(* CODESYS project Traslo_st_UBICA_POR_COLOR_y_ROBOT+TABLA-.project
   CompiledLibraryCompatibilityVersion: CODESYS V3.5 SP16 Patch 4

Project tree, tasks and I/O mapping:
  Device : CODESYS Control Win V3 x64, 3S - Smart Software Solutions GmbH, version 3.5.16.40
    application Application
      libraries: Standard, * (System); VisuDialogs, * (System); CmpBitmapPool, * (System)
      task VISU_TASK (cyclic, interval 100 ms, priority 31) calls VisuElems.Visu_Prg
      task MainTask (cyclic, interval t#20ms, priority 1) calls PLC_PRG
      program ANALOGICAS [LD]
      Symbols
      program PLC_PRG [ST]
      visualisation Panel_control
      global variables GVL
      function block ESCALADO [FBD]
      image pool ImagePool
  libraries: Util, * (System); Net Base Services, 3.5.19.20 (3S - Smart Software Solutions GmbH)
  5ce3da45-db07-42e7-a21c-a00fff4ed8f6|C:\Users\GGARCES\OneDrive - congeladosnavarra.com\ICONOS\scada\SETA_EMERG_ON.png
  text list GlobalTextList
  5ce3da45-db07-42e7-a21c-a00fff4ed8f6|C:\Users\GGARCES\OneDrive - congeladosnavarra.com\ICONOS\scada\SETA_EMERG_OFF.png
*)

// Device/Application/GVL
{attribute 'qualified_only'}
VAR_GLOBAL
	VISION_AZUL : BOOL;
	VISION_VERDE : BOOL;
	VISION_METAL : BOOL;
	NUMERO_ESTANTE : REAL;
	POSICION : REAL;
	x_position : REAL;                          //max 9 posiciones
	Z_position : REAL;
	X_position_FILTRADA: REAL;
	Z_position_FILTRADA: REAL;
END_VAR

// Device/Application/PLC_PRG
PROGRAM PLC_PRG
VAR
	Tim_carga : TON ; 
	sys_on: BOOL;
	sys_auto: BOOL;
	sys_man: BOOL;
	count : INT;
	count_forks: INT;
	flanco_carga: BOOL;flanco_forks_out: BOOL;
	R_TRIG1: R_trig;R_TRIG : R_TRIG;
	R_TRIG_ESTANTE : R_TRIG;
	CTU_MOV: CTU;
	TIM_POSICION: TOF;
	Tim_descarga: TON;
	TRASLO_CARGADO: BOOL;
	TIM_POS0: TON;
	Tim_descarga1: TON;
	PALET_POS: BOOL;
	Tim_descarga2: TON;
	Tim_descarga3: TON;
	Tim_descarga4: TON;
	Tim_descarga5: TON;
	R_TRIG_AZUL: R_TRIG;
	R_TRIG_VERDE: R_TRIG;
	R_TRIG_METAL: R_TRIG;
	CTU_AZUL: CTU;
	CTU_VERDE : CTU;
	CTU_METAL : CTU;
	CNT_TOTAL : CTU;
	CNT_PIEZAS : CTU;
	// color verde
	pos1 : BOOL;
	pos2 : BOOL;
	pos3 : BOOL;
	pos4 : BOOL;
	pos5 : BOOL;
	pos6 : BOOL;
	pos7 : BOOL;
	pos8 : BOOL;
	pos9 : BOOL;
	pos10 : BOOL;
	pos11 : BOOL;
	pos12 : BOOL;	
    pos13 : BOOL;
	pos14 : BOOL;
	pos15 : BOOL;
	pos16 : BOOL;
	pos17 : BOOL;
	pos18 : BOOL;
	// color azul
	pos19 : BOOL;
	pos20 : BOOL;
	pos21 : BOOL;
	pos22 : BOOL;
	pos23 : BOOL;
	pos24 : BOOL;
	pos25 : BOOL;
	pos26 : BOOL;
	pos27 : BOOL;
	pos28 : BOOL;
	pos29 : BOOL;
	pos30 : BOOL;	
    pos31 : BOOL;
	pos32 : BOOL;
	pos33 : BOOL;
	pos34 : BOOL;
	pos35 : BOOL;
	pos36 : BOOL;
	// color metal
	pos37 : BOOL;
	pos38 : BOOL;
	pos39 : BOOL;
	pos40 : BOOL;
	pos41 : BOOL;
	pos42 : BOOL;
	pos43 : BOOL;
	pos44 : BOOL;
	pos45 : BOOL;
	pos46 : BOOL;
	pos47 : BOOL;
	pos48 : BOOL;	
    pos49 : BOOL;
	pos50 : BOOL;
	pos51 : BOOL;
	pos52 : BOOL;
	pos53 : BOOL;
	pos54 : BOOL;
	
	color_verde_saturado : BOOL;
	color_azul_saturado : BOOL;
	color_metal_saturado : BOOL;
	SENSOR0_0: BOOL;
	TON_bajar1 : ton ;
	TON_subir1 : ton ;
	TON_bajar2 : ton ;
	TON_subir2 : ton ;
	TON_avanzar : ton ;
	TON_retroceder : ton ;
	TON_reset: ton;
	fin_ciclo_robot_cartesiano : BOOL ;
	a: BOOL;
	bit1 : INT ;
	CONTADOR_TOTAL: WORD;
	REGISTRO: ARRAY [1..55] OF WORD;
	POS: word;
	STARTFP: r_trig;
END_VAR
VAR_INPUT
	At_entry : BOOL;
	At_exit : BOOL;
	At_load : BOOL;
	At_unload : BOOL;
	SENSOR_0: BOOL;
	SENSOR_1: BOOL;
	auto : BOOL;
	Emergency_stop : BOOL;
	Manual : BOOL;
	limit_right : BOOL;
	limit_left : BOOL;
	Reset : BOOL;
	Start : BOOL;
	Stop : BOOL;
	stacker_crane_limit_right : BOOL;
	stacker_crane_limit_left : BOOL;
	stacker_crane_limit_middle : BOOL;
	MANDAR_POSICION : BOOL;
	GO: BOOL;
	RESET_NUMERO_ESTANTE : BOOL;
	SENSOR_piezas_cinta :BOOL;
	robot_ocupado : BOOL;
	FALLO_ROBOT : BOOL;
	detec_piezas_cartesiano : BOOL ;
	deteccion_pieza_robot_cart: BOOL;
END_VAR

VAR_OUTPUT
	//rodillos
	Emitter : BOOL;
	RODILLOS_1: BOOL;
	CURVA_RODILLOS_2: BOOL;
	RODILLOS_3: BOOL;
	Entry_CONVEYOR_3 : BOOL;
	Load_conveyor_4 : BOOL;
	Exit_conveyor : BOOL;
	UnLoad_conveyor_4 : BOOL;
	Remover : BOOL;
	
	Forks_left : BOOL;
	Forks_right : BOOL;
	// luces
	Reset_light : BOOL;
	Start_light : BOOL;
	Stop_light : BOOL;
	
	stacker_crane_x_sp : REAL;
	stacker_crane_z_sp : REAL;
	ALARMA_ACTIVA : BOOL;
	
	Emisor_piezas : BOOL;
	cinta_piezas : BOOL;
	ON_ROBOT : BOOL ;
	
	bajar_robot_cartesiano : BOOL;
	subir_robot_cartesiano : BOOL;
	agarrar_pieza_robot_cart : BOOL ;
	avanzar_robot_cartesiano : BOOL ;
	
	CINTA_PIEZAS_ACABADAS : BOOL ;
	TOPE_PIEZAS : BOOL ;
END_VAR


ANALOGICAS ();

// PROGRAMA PARA SIMULAR CON FACTORY IO UN TRASLO

//emergencia
IF NOT Emergency_stop OR NOT Stop THEN
	sys_on := FALSE;
	sys_auto:= FALSE;
	Entry_CONVEYOR_3 := FALSE;
	Load_conveyor_4 := FALSE;
	Forks_left := FALSE;
	Forks_right := FALSE;
	stacker_crane_x_sp := 0;
    stacker_crane_z_sp := 0;
	TRASLO_CARGADO := FALSE;
	COUNT_FORKS := 0;
	gvl.Z_position := 0;
	gvl.x_position := 0;
	PALET_POS := FALSE;
	GVL.POSICION := 0;
	pos1 := 0;pos2 := 0;pos3 := 0;pos4 := 0;pos5 := 0;pos6 := 0;pos7 := 0;pos8 := 0;pos9 := 0;pos10:= 0;
	pos11:= 0;pos12:= 0;pos13:= 0;pos14:= 0;pos15:= 0;pos16:= 0;pos17:= 0;pos18:= 0;pos19:= 0;pos20:= 0;
	pos21:= 0;pos22:= 0;pos23:= 0;pos24:= 0;pos25:= 0;pos26:= 0;pos27:= 0;pos28:= 0;pos29:= 0;pos30:= 0;
	pos31:= 0;pos32:= 0;pos33:= 0;pos34:= 0;pos35:= 0;pos36:= 0;pos37:= 0;pos38:= 0;pos39:= 0;pos40:= 0;
	pos41:= 0;pos42:= 0;pos43:= 0;pos44:= 0;pos45:= 0;pos46:= 0;pos47:= 0;pos48:= 0;pos49:= 0;pos50:= 0;
	pos51:= 0;pos52:= 0;pos53:= 0;pos54:= 0;
	POS:=0;
    
END_IF

// FALLO POSICION 0 EN FACTORY I/O FILTRO PARA QUE FUNCIONE BIEN
IF gvl.X_position_FILTRADA <0 THEN gvl.X_position_FILTRADA :=0;
IF gvl.Z_position_FILTRADA <0 THEN gvl.Z_position_FILTRADA :=0;	
END_IF
END_IF

// On
IF Start AND auto THEN
	sys_on := TRUE;
	stacker_crane_x_sp := 0;
    stacker_crane_z_sp := 0;
END_IF

//Auto
IF sys_on AND auto THEN
	sys_auto:= TRUE;
	sys_man := FALSE;
END_IF

// Manual
IF sys_on AND manual THEN
	sys_auto:= FALSE;
	sys_man := TRUE;
END_IF

// Reset
IF reset  THEN
	count:= 0;
	count_forks := 0;
	stacker_crane_x_sp := 0;
    stacker_crane_z_sp := 0;
	GVL.POSICION := 0;
END_IF

IF RESET AND NOT stacker_crane_limit_middle AND stacker_crane_limit_left THEN Forks_right := TRUE; END_IF
IF RESET AND NOT stacker_crane_limit_middle AND stacker_crane_limit_right THEN Forks_left := TRUE; END_IF 
IF RESET AND stacker_crane_limit_middle THEN 
	Forks_right := FALSE;
	Forks_left := FALSE;
    PALET_POS := FALSE;	
END_IF

// EMISOR DE PALETS
IF SYS_ON AND SENSOR_0 AND NOT ALARMA_ACTIVA THEN
	Emitter := TRUE;
END_IF
IF Emitter AND NOT SENSOR_0 OR NOT SYS_ON THEN
	Emitter := false;
END_IF
// Caminos de rodillos 1
IF sys_auto AND bit1 = 8 AND CURVA_RODILLOS_2  AND NOT ALARMA_ACTIVA AND NOT Emitter THEN
	RODILLOS_1 := TRUE;
END_IF	
IF sys_auto AND NOT CURVA_RODILLOS_2 OR Emitter OR  ALARMA_ACTIVA THEN
	RODILLOS_1 := FALSE;
END_IF
// Curva de rodillos 2
IF sys_auto AND RODILLOS_3 AND NOT ALARMA_ACTIVA THEN
	CURVA_RODILLOS_2 := TRUE;
IF sys_auto AND NOT SENSOR_1 AND NOT ALARMA_ACTIVA OR NOT RODILLOS_3 THEN
	CURVA_RODILLOS_2 := FALSE;
END_IF
END_IF
// Caminos de rodillos 3
IF sys_auto AND Entry_CONVEYOR_3 AND NOT ALARMA_ACTIVA THEN
	RODILLOS_3 := TRUE;
END_IF
IF sys_auto AND NOT at_entry AND NOT ALARMA_ACTIVA OR NOT Entry_CONVEYOR_3 THEN
    RODILLOS_3 := FALSE;
END_IF
// Entry conveyor 3
IF sys_auto AND Load_conveyor_4 AND NOT ALARMA_ACTIVA THEN
	Entry_CONVEYOR_3 := TRUE;
END_IF
IF sys_auto AND NOT at_load AND NOT ALARMA_ACTIVA OR NOT Load_conveyor_4 THEN
    Entry_CONVEYOR_3 := FALSE;
END_IF
// load conveyor 4
IF sys_auto AND at_load AND NOT ALARMA_ACTIVA THEN
	Load_conveyor_4 := TRUE;
ELSE
	Load_conveyor_4 := FALSE;	
END_IF

// Flanco contador palets a traslo
    R_TRIG(CLK:= NOT At_load, Q=> flanco_carga); 

// Llamada a traslo y asigna posicion 
IF FLANCO_CARGA THEN
	Entry_CONVEYOR_3 := FALSE;
	Load_conveyor_4 := FALSE;
END_IF
// TIEMPO EN POSICION DE INICIO
	TIM_POS0(IN := gvl.x_position_FILTRADA < 0.1 AND gvl.Z_position_FILTRADA =0 AND NOT AT_LOAD , PT:= T#1S); 
	IF TIM_POS0.Q THEN
	PALET_POS := TRUE;
	else
	PALET_POS:= FALSE;
	END_IF

// CONTROL DE PALETS POR PRODUCTO -----COLOR------

R_TRIG_AZUL(CLK:= GVL.VISION_AZUL);
R_TRIG_VERDE(CLK:= GVL.VISION_VERDE);
R_TRIG_METAL(CLK:= GVL.VISION_METAL);

CTU_AZUL(CU:= R_TRIG_AZUL.CLK, RESET:=RESET OR NOT Emergency_stop);
CTU_VERDE(CU:= R_TRIG_VERDE.CLK, RESET:=RESET OR NOT Emergency_stop);
CTU_METAL(CU:= R_TRIG_METAL.CLK, RESET:=RESET OR NOT Emergency_stop);

//AZUL
IF R_TRIG_AZUL.CLK THEN 
	GVL.POSICION := CTU_AZUL.CV;
END_IF
//VERDE
IF R_TRIG_VERDE.CLK THEN 
	GVL.POSICION := CTU_VERDE.CV + 18;
END_IF
//METAL
IF R_TRIG_METAL.CLK THEN 
	GVL.POSICION := CTU_METAL.CV + 36;
END_IF
// ------------ COGER PALET ---------------
// salida uñas
IF PALET_POS AND stacker_crane_limit_middle THEN
	Forks_left := TRUE;
END_IF

IF flanco_forks_out THEN
	count_forks := count_forks + 1;
END_IF

//FLANCO_UÑAS CARGA FUERA
R_TRIG1(CLK:=Forks_left AND NOT stacker_crane_limit_middle, Q=> flanco_forks_out); 

// RETARDO RECOGIDA UÑAS
Tim_carga(IN := stacker_crane_limit_left, PT:= T#1S); 

// elevar coger palet
IF stacker_crane_limit_left AND sys_auto AND stacker_crane_x_sp = 0 (*atras*)THEN
	stacker_crane_z_sp :=0.30;
END_IF

// uñas atras
IF stacker_crane_limit_left AND stacker_crane_z_sp >= 0.3 AND Tim_carga.Q THEN
	Forks_left := FALSE;
	TRASLO_CARGADO := TRUE;
	PALET_POS := FALSE;
END_IF 

// contador de palets en el traslo     
CTU_MOV(CU:= stacker_crane_limit_middle AND count_forks = 1 AND NOT MANDAR_POSICION AND NOT GO, RESET:=RESET OR RESET_NUMERO_ESTANTE OR NOT Emergency_stop, PV:= 100); 
CNT_TOTAL(CU:= count_forks = 1,RESET:= RESET AND NOT Emergency_stop,PV:= 55);
//
TIM_POSICION(IN := count_forks = 1 AND stacker_crane_limit_middle, PT:= T#200S); 
// RESET CONTADOR CUANDO ELIGES ESTANTERIA EN MANUAL
R_TRIG_ESTANTE (CLK:= RESET_NUMERO_ESTANTE );

//-----------------------------------------------------------------------------


//------------ PRIMERA FILA --------------------------


//-----------------------------------------------------------------------------
// POSICION 1
IF GVL.POSICION = 1 AND count_forks=1 AND stacker_crane_limit_middle AND TIM_POSICION.Q THEN
     stacker_crane_x_sp := 1.06;
     stacker_crane_z_sp := 0.8;
END_IF
// dejar carga posicion 1
IF GVL.POSICION = 1 AND TIM_POSICION.Q AND count_forks=1 AND gvl.x_position_FILTRADA < 0.98 AND gvl.x_position_FILTRADA > 0.96 AND gvl.Z_position_FILTRADA < 0.8 AND gvl.Z_position_FILTRADA > 0.7 THEN 
    Forks_right := TRUE;	
IF stacker_crane_limit_right THEN
	stacker_crane_z_sp := 0.4;
END_IF	
END_IF
//-----------------------------------------------------------------------------

// POSICION 2
IF GVL.POSICION = 2 AND count_forks=1 AND stacker_crane_limit_middle AND TIM_POSICION.Q THEN
	 stacker_crane_x_sp := 2.14;
     stacker_crane_z_sp := 0.8;
END_IF 
// dejar carga posicion 2
IF GVL.POSICION = 2 AND TIM_POSICION.Q AND count_forks=1 AND gvl.x_position_FILTRADA < 2.07 AND gvl.x_position_FILTRADA > 2.05 AND gvl.Z_position_FILTRADA < 0.8 AND gvl.Z_position_FILTRADA > 0.7 THEN 
    Forks_right := TRUE;
IF stacker_crane_limit_right THEN
	stacker_crane_z_sp := 0.4;
END_IF	
END_IF

//-----------------------------------------------------------------------------
// POSICION 3
IF GVL.POSICION = 3 AND count_forks=1 AND stacker_crane_limit_middle AND TIM_POSICION.Q THEN
	  stacker_crane_x_sp := 3.21;
     stacker_crane_z_sp := 0.8;
END_IF 
// dejar carga posicion 3
IF GVL.POSICION = 3 AND TIM_POSICION.Q AND count_forks=1 AND gvl.x_position < 3.22 AND gvl.x_position > 3.20 AND gvl.Z_position < 0.8 AND gvl.Z_position > 0.7 THEN 
    Forks_right := TRUE;
IF stacker_crane_limit_right THEN
	stacker_crane_z_sp := 0.4;
END_IF	
END_IF  
//-----------------------------------------------------------------------------

// POSICION 4
IF GVL.POSICION = 4 AND count_forks=1 AND stacker_crane_limit_middle AND TIM_POSICION.Q THEN
	  stacker_crane_x_sp := 4.28;
     stacker_crane_z_sp := 0.8;
	 END_IF
// dejar carga posicion 4
IF GVL.POSICION = 4 AND TIM_POSICION.Q AND count_forks=1 AND gvl.x_position < 4.29 AND gvl.x_position > 4.27 AND gvl.Z_position < 0.8 AND gvl.Z_position > 0.7 THEN 
    Forks_right := TRUE;
IF stacker_crane_limit_right THEN
	stacker_crane_z_sp := 0.4;
	
END_IF  
END_IF 
//-----------------------------------------------------------------------------
// POSICION 5
IF GVL.POSICION = 5 AND count_forks=1 AND stacker_crane_limit_middle AND TIM_POSICION.Q THEN
	  stacker_crane_x_sp := 5.36;
     stacker_crane_z_sp := 0.8;
END_IF 
// dejar carga posicion 5
IF GVL.POSICION = 5 AND TIM_POSICION.Q AND count_forks=1 AND gvl.x_position < 5.37 AND gvl.x_position > 5.35 AND gvl.Z_position < 0.8 AND gvl.Z_position > 0.7 THEN 
    Forks_right := TRUE;
IF stacker_crane_limit_right THEN
	stacker_crane_z_sp := 0.4;	
END_IF  
END_IF
//-----------------------------------------------------------------------------
// POSICION 6
IF GVL.POSICION = 6 AND count_forks=1 AND stacker_crane_limit_middle AND TIM_POSICION.Q THEN
	  stacker_crane_x_sp := 6.45;
     stacker_crane_z_sp := 0.8;
END_IF 
// dejar carga posicion 6
IF GVL.POSICION = 6 AND TIM_POSICION.Q AND count_forks=1 AND gvl.x_position < 6.46 AND gvl.x_position > 6.44 AND gvl.Z_position < 0.9 AND gvl.Z_position > 0.7 THEN 
    Forks_right := TRUE;
IF stacker_crane_limit_right THEN
	stacker_crane_z_sp := 0.4;
END_IF  
END_IF 
//-----------------------------------------------------------------------------
// POSICION 7
IF GVL.POSICION = 7 AND count_forks=1 AND stacker_crane_limit_middle AND TIM_POSICION.Q THEN
	  stacker_crane_x_sp := 7.52;
     stacker_crane_z_sp := 0.8;
END_IF 
// dejar carga posicion 7
IF GVL.POSICION = 7 AND TIM_POSICION.Q AND count_forks=1 AND gvl.x_position < 7.53 AND gvl.x_position > 7.51 AND gvl.Z_position < 0.9 AND gvl.Z_position > 0.7 THEN 
    Forks_right := TRUE;
IF stacker_crane_limit_right THEN
	stacker_crane_z_sp := 0.4;
END_IF	
END_IF  
//-----------------------------------------------------------------------------
// POSICION 8
IF GVL.POSICION = 8 AND count_forks=1 AND stacker_crane_limit_middle AND TIM_POSICION.Q THEN
	  stacker_crane_x_sp := 8.59;
     stacker_crane_z_sp := 0.8;
END_IF 
// dejar carga posicion 8
IF GVL.POSICION = 8 AND TIM_POSICION.Q AND count_forks=1 AND gvl.x_position < 8.60 AND gvl.x_position > 8.58 AND gvl.Z_position < 0.9 AND gvl.Z_position > 0.7 THEN 
    Forks_right := TRUE;
IF stacker_crane_limit_right THEN
	stacker_crane_z_sp := 0.4;
END_IF	
END_IF  
//-----------------------------------------------------------------------------
// POSICION 9
IF GVL.POSICION = 9 AND count_forks=1 AND stacker_crane_limit_middle AND TIM_POSICION.Q THEN
	  stacker_crane_x_sp := 9.66;
     stacker_crane_z_sp := 0.8;
END_IF 
// dejar carga posicion 9
IF GVL.POSICION = 9 AND TIM_POSICION.Q AND count_forks=1 AND gvl.x_position > 9.65 AND gvl.x_position < 9.67 AND gvl.Z_position < 0.9 AND gvl.Z_position > 0.7 THEN 
    Forks_right := TRUE;
IF stacker_crane_limit_right THEN
	stacker_crane_z_sp := 0.4;
END_IF	
END_IF  
//-----------------------------------------------------------------------------

// --------- SEGUNDA FILA --------------


//-----------------------------------------------------------------------------

// POSICION 10
IF GVL.POSICION = 10 AND count_forks=1 AND stacker_crane_limit_middle AND TIM_POSICION.Q  THEN
	  stacker_crane_x_sp := 1.06;
      stacker_crane_z_sp := 2.50;
END_IF 
// dejar carga posicion 10
IF GVL.POSICION = 10 AND TIM_POSICION.Q AND count_forks=1 AND gvl.x_position < 1.07 AND gvl.x_position > 1.05 AND gvl.Z_position < 2.51 AND gvl.Z_position > 2.49 THEN 
    Forks_right := TRUE;
IF stacker_crane_limit_right THEN
	stacker_crane_z_sp := 2.0;
END_IF	
END_IF  
//-----------------------------------------------------------------------------

// POSICION 11
IF GVL.POSICION = 11 AND count_forks=1 AND stacker_crane_limit_middle AND TIM_POSICION.Q  THEN
	  stacker_crane_x_sp := 2.15;
      stacker_crane_z_sp := 2.5;
END_IF 
// dejar carga posicion 11
IF GVL.POSICION = 11 AND TIM_POSICION.Q AND count_forks=1 AND gvl.x_position < 2.16 AND gvl.x_position > 2.14 AND gvl.Z_position < 2.51 AND gvl.Z_position > 2.49 THEN 
    Forks_right := TRUE;
IF stacker_crane_limit_right THEN
	stacker_crane_z_sp := 2.0;
END_IF	
END_IF  
//-----------------------------------------------------------------------------

// POSICION 12
IF GVL.POSICION = 12 AND count_forks=1 AND stacker_crane_limit_middle AND TIM_POSICION.Q  THEN
	  stacker_crane_x_sp := 3.21;
      stacker_crane_z_sp := 2.5;
END_IF 
// dejar carga posicion 12
IF GVL.POSICION = 12 AND TIM_POSICION.Q AND count_forks=1 AND gvl.x_position < 3.22 AND gvl.x_position > 3.20 AND gvl.Z_position < 2.51 AND gvl.Z_position > 2.49 THEN 
    Forks_right := TRUE;
IF stacker_crane_limit_right THEN
	stacker_crane_z_sp := 2.0;
END_IF	
END_IF  
//-----------------------------------------------------------------------------

// POSICION 13
IF GVL.POSICION = 13 AND count_forks=1 AND stacker_crane_limit_middle AND TIM_POSICION.Q  THEN
	  stacker_crane_x_sp := 4.28;
      stacker_crane_z_sp := 2.5;
END_IF 
// dejar carga posicion 13
IF GVL.POSICION = 13 AND TIM_POSICION.Q AND count_forks=1 AND gvl.x_position < 4.29 AND gvl.x_position > 4.27 AND gvl.Z_position < 2.51 AND gvl.Z_position > 2.49 THEN 
    Forks_right := TRUE;
IF stacker_crane_limit_right THEN
	stacker_crane_z_sp := 2.0;
END_IF	
END_IF  
//-----------------------------------------------------------------------------

// POSICION 14
IF GVL.POSICION = 14 AND count_forks=1 AND stacker_crane_limit_middle AND TIM_POSICION.Q  THEN
	  stacker_crane_x_sp := 5.36;
      stacker_crane_z_sp := 2.5;
END_IF 
// dejar carga posicion 14
IF GVL.POSICION = 14 AND TIM_POSICION.Q AND count_forks=1 AND gvl.x_position < 5.37 AND gvl.x_position > 5.35 AND gvl.Z_position < 2.51 AND gvl.Z_position > 2.49 THEN 
    Forks_right := TRUE;
IF stacker_crane_limit_right THEN
	stacker_crane_z_sp := 2.0;
END_IF	
END_IF  
//-----------------------------------------------------------------------------

// POSICION 15
IF GVL.POSICION = 15 AND count_forks=1 AND stacker_crane_limit_middle AND TIM_POSICION.Q  THEN
	  stacker_crane_x_sp := 6.45;
      stacker_crane_z_sp := 2.5;
END_IF 
// dejar carga posicion 15
IF GVL.POSICION = 15 AND TIM_POSICION.Q AND count_forks=1 AND gvl.x_position < 6.46 AND gvl.x_position > 6.44 AND gvl.Z_position < 2.51 AND gvl.Z_position > 2.49 THEN 
    Forks_right := TRUE;
IF stacker_crane_limit_right THEN
	stacker_crane_z_sp := 2.0;
END_IF	
END_IF  
//-----------------------------------------------------------------------------

// POSICION 16
IF GVL.POSICION = 16 AND count_forks=1 AND stacker_crane_limit_middle AND TIM_POSICION.Q  THEN
	  stacker_crane_x_sp := 7.52;
      stacker_crane_z_sp := 2.5;
END_IF 
// dejar carga posicion 16
IF GVL.POSICION = 16 AND TIM_POSICION.Q AND count_forks=1 AND gvl.x_position < 7.53 AND gvl.x_position > 7.51 AND gvl.Z_position < 2.51 AND gvl.Z_position > 2.49 THEN 
    Forks_right := TRUE;
IF stacker_crane_limit_right THEN
	stacker_crane_z_sp := 2.0;
END_IF	
END_IF  
//-----------------------------------------------------------------------------

// POSICION 17
IF GVL.POSICION = 17 AND count_forks=1 AND stacker_crane_limit_middle AND TIM_POSICION.Q  THEN
	  stacker_crane_x_sp := 8.59;
      stacker_crane_z_sp := 2.5;
END_IF 
// dejar carga posicion 17
IF GVL.POSICION = 17 AND TIM_POSICION.Q AND count_forks=1 AND gvl.x_position < 8.60 AND gvl.x_position > 8.58 AND gvl.Z_position < 2.51 AND gvl.Z_position > 2.49 THEN 
    Forks_right := TRUE;
IF stacker_crane_limit_right THEN
	stacker_crane_z_sp := 2.0;
END_IF	
END_IF  
//-----------------------------------------------------------------------------

// POSICION 18
IF GVL.POSICION = 18 AND count_forks=1 AND stacker_crane_limit_middle AND TIM_POSICION.Q  THEN
	  stacker_crane_x_sp := 9.66;
      stacker_crane_z_sp := 2.5;
END_IF 
// dejar carga posicion 18
IF GVL.POSICION = 18 AND TIM_POSICION.Q AND count_forks=1 AND gvl.x_position < 9.67 AND gvl.x_position > 9.65 AND gvl.Z_position < 2.51 AND gvl.Z_position > 2.49 THEN 
    Forks_right := TRUE;
IF stacker_crane_limit_right THEN
	stacker_crane_z_sp := 2.0;
END_IF	
END_IF  
//-----------------------------------------------------------------------------  

// --------- TERCERA FILA --------------

//-----------------------------------------------------------------------------
// POSICION 19
IF GVL.POSICION = 19 AND count_forks=1 AND stacker_crane_limit_middle AND TIM_POSICION.Q  THEN
	  stacker_crane_x_sp := 1.06;
      stacker_crane_z_sp := 4.20;
END_IF 
// dejar carga posicion 19
IF GVL.POSICION = 19 AND TIM_POSICION.Q AND count_forks=1 AND gvl.x_position < 1.07 AND gvl.x_position > 1.05 AND gvl.Z_position < 4.21 AND gvl.Z_position > 4.19 THEN 
    Forks_right := TRUE;
IF stacker_crane_limit_right THEN
	stacker_crane_z_sp := 3.90;
END_IF	
END_IF  
//-----------------------------------------------------------------------------

// POSICION 20
IF GVL.POSICION = 20 AND count_forks=1 AND stacker_crane_limit_middle AND TIM_POSICION.Q  THEN
	  stacker_crane_x_sp := 2.15;
      stacker_crane_z_sp := 4.20;
END_IF 
// dejar carga posicion 20
IF GVL.POSICION = 20 AND TIM_POSICION.Q AND count_forks=1 AND gvl.x_position < 2.16 AND gvl.x_position > 2.14 AND gvl.Z_position < 4.21 AND gvl.Z_position > 4.19 THEN 
    Forks_right := TRUE;
IF stacker_crane_limit_right THEN
	stacker_crane_z_sp := 3.90;
END_IF	
END_IF  
//-----------------------------------------------------------------------------

// POSICION 21
IF GVL.POSICION = 21 AND count_forks=1 AND stacker_crane_limit_middle AND TIM_POSICION.Q  THEN
	  stacker_crane_x_sp := 3.21;
      stacker_crane_z_sp := 4.20;
END_IF 
// dejar carga posicion 21
IF GVL.POSICION = 21 AND TIM_POSICION.Q AND count_forks=1 AND gvl.x_position < 3.22 AND gvl.x_position > 3.20 AND gvl.Z_position < 4.21 AND gvl.Z_position > 4.19 THEN 
    Forks_right := TRUE;
IF stacker_crane_limit_right THEN
	stacker_crane_z_sp := 3.90;
END_IF	
END_IF  
//-----------------------------------------------------------------------------

// POSICION 22
IF GVL.POSICION = 22 AND count_forks=1 AND stacker_crane_limit_middle AND TIM_POSICION.Q  THEN
	  stacker_crane_x_sp := 4.29;
      stacker_crane_z_sp := 4.20;
END_IF 
// dejar carga posicion 22
IF GVL.POSICION = 22 AND TIM_POSICION.Q AND count_forks=1 AND gvl.x_position < 4.30 AND gvl.x_position > 4.28 AND gvl.Z_position < 4.21 AND gvl.Z_position > 4.19 THEN 
    Forks_right := TRUE;
IF stacker_crane_limit_right THEN
	stacker_crane_z_sp := 3.90;
END_IF	
END_IF  
//-----------------------------------------------------------------------------

// POSICION 23
IF GVL.POSICION = 23 AND count_forks=1 AND stacker_crane_limit_middle AND TIM_POSICION.Q  THEN
	  stacker_crane_x_sp := 5.36;
      stacker_crane_z_sp := 4.20;
END_IF 
// dejar carga posicion 23
IF GVL.POSICION = 23 AND TIM_POSICION.Q AND count_forks=1 AND gvl.x_position < 5.37 AND gvl.x_position > 5.35 AND gvl.Z_position < 4.21 AND gvl.Z_position > 4.19 THEN 
    Forks_right := TRUE;
IF stacker_crane_limit_right THEN
	stacker_crane_z_sp := 3.90;
END_IF	
END_IF  
//-----------------------------------------------------------------------------

// POSICION 24
IF GVL.POSICION = 24 AND count_forks=1 AND stacker_crane_limit_middle AND TIM_POSICION.Q  THEN
	  stacker_crane_x_sp := 6.44;
      stacker_crane_z_sp := 4.20;
END_IF 
// dejar carga posicion 24
IF GVL.POSICION = 24 AND TIM_POSICION.Q AND count_forks=1 AND gvl.x_position < 6.45 AND gvl.x_position > 6.43 AND gvl.Z_position < 4.21 AND gvl.Z_position > 4.19 THEN 
    Forks_right := TRUE;
IF stacker_crane_limit_right THEN
	stacker_crane_z_sp := 3.90;
END_IF	
END_IF  
//-----------------------------------------------------------------------------

// POSICION 25
IF GVL.POSICION = 25 AND count_forks=1 AND stacker_crane_limit_middle AND TIM_POSICION.Q  THEN
	  stacker_crane_x_sp := 7.51;
      stacker_crane_z_sp := 4.20;
END_IF 
// dejar carga posicion 25
IF GVL.POSICION = 25 AND TIM_POSICION.Q AND count_forks=1 AND gvl.x_position < 7.52 AND gvl.x_position > 7.50 AND gvl.Z_position < 4.21 AND gvl.Z_position > 4.19 THEN 
    Forks_right := TRUE;
IF stacker_crane_limit_right THEN
	stacker_crane_z_sp := 3.90;
END_IF	
END_IF  
//-----------------------------------------------------------------------------

// POSICION 26
IF GVL.POSICION = 26 AND count_forks=1 AND stacker_crane_limit_middle AND TIM_POSICION.Q  THEN
	  stacker_crane_x_sp := 8.59;
      stacker_crane_z_sp := 4.20;
END_IF 
// dejar carga posicion 26
IF GVL.POSICION = 26 AND TIM_POSICION.Q AND count_forks=1 AND gvl.x_position < 8.60 AND gvl.x_position > 8.58 AND gvl.Z_position < 4.21 AND gvl.Z_position > 4.19 THEN 
    Forks_right := TRUE;
IF stacker_crane_limit_right THEN
	stacker_crane_z_sp := 3.90;
END_IF	
END_IF  
//-----------------------------------------------------------------------------

// POSICION 27
IF GVL.POSICION = 27 AND count_forks=1 AND stacker_crane_limit_middle AND TIM_POSICION.Q  THEN
	  stacker_crane_x_sp := 9.66;
      stacker_crane_z_sp := 4.20;
END_IF 
// dejar carga posicion 27
IF GVL.POSICION = 27 AND TIM_POSICION.Q AND count_forks=1 AND gvl.x_position < 9.67 AND gvl.x_position > 9.65 AND gvl.Z_position < 4.21 AND gvl.Z_position > 4.19 THEN 
    Forks_right := TRUE;
IF stacker_crane_limit_right THEN
	stacker_crane_z_sp := 3.90;
END_IF	
END_IF  
//-----------------------------------------------------------------------------  


// --------- CUARTA FILA --------------

//-----------------------------------------------------------------------------
// POSICION 28
IF GVL.POSICION = 28 AND count_forks=1 AND stacker_crane_limit_middle AND TIM_POSICION.Q  THEN
	  stacker_crane_x_sp := 1.06;
      stacker_crane_z_sp := 5.66;
END_IF 
// dejar carga posicion 28
IF GVL.POSICION = 28 AND TIM_POSICION.Q AND count_forks=1 AND gvl.x_position < 1.07 AND gvl.x_position > 1.05 AND gvl.Z_position < 5.67 AND gvl.Z_position > 5.65 THEN 
    Forks_right := TRUE;
IF stacker_crane_limit_right THEN
	stacker_crane_z_sp := 5.40;
END_IF	
END_IF  
//-----------------------------------------------------------------------------

// POSICION 29
IF GVL.POSICION = 29 AND count_forks=1 AND stacker_crane_limit_middle AND TIM_POSICION.Q  THEN
	  stacker_crane_x_sp := 2.15;
      stacker_crane_z_sp := 5.66;
END_IF 
// dejar carga posicion 29
IF GVL.POSICION = 29 AND TIM_POSICION.Q AND count_forks=1 AND gvl.x_position < 2.16 AND gvl.x_position > 2.14 AND gvl.Z_position < 5.67 AND gvl.Z_position > 5.65 THEN 
    Forks_right := TRUE;
IF stacker_crane_limit_right THEN
	stacker_crane_z_sp := 5.40;
END_IF	
END_IF  
//-----------------------------------------------------------------------------

// POSICION 30
IF GVL.POSICION = 30 AND count_forks=1 AND stacker_crane_limit_middle AND TIM_POSICION.Q  THEN
	  stacker_crane_x_sp := 3.21;
      stacker_crane_z_sp := 5.66;
END_IF 
// dejar carga posicion 30
IF GVL.POSICION = 30 AND TIM_POSICION.Q AND count_forks=1 AND gvl.x_position < 3.22 AND gvl.x_position > 3.20 AND gvl.Z_position < 5.67 AND gvl.Z_position > 5.65 THEN 
    Forks_right := TRUE;
IF stacker_crane_limit_right THEN
	stacker_crane_z_sp := 5.40;
END_IF	
END_IF  
//-----------------------------------------------------------------------------

// POSICION 31
IF GVL.POSICION = 31 AND count_forks=1 AND stacker_crane_limit_middle AND TIM_POSICION.Q  THEN
	  stacker_crane_x_sp := 4.29;
      stacker_crane_z_sp := 5.66;
END_IF 
// dejar carga posicion 31
IF GVL.POSICION = 31 AND TIM_POSICION.Q AND count_forks=1 AND gvl.x_position < 4.30 AND gvl.x_position > 4.28 AND gvl.Z_position < 5.67 AND gvl.Z_position > 5.65 THEN 
    Forks_right := TRUE;
IF stacker_crane_limit_right THEN
	stacker_crane_z_sp := 5.40;
END_IF	
END_IF  
//-----------------------------------------------------------------------------

// POSICION 32
IF GVL.POSICION = 32 AND count_forks=1 AND stacker_crane_limit_middle AND TIM_POSICION.Q  THEN
	  stacker_crane_x_sp := 5.36;
      stacker_crane_z_sp := 5.66;
END_IF 
// dejar carga posicion 32
IF GVL.POSICION = 32 AND TIM_POSICION.Q AND count_forks=1 AND gvl.x_position < 5.37 AND gvl.x_position > 5.35 AND gvl.Z_position < 5.67 AND gvl.Z_position > 5.65 THEN 
    Forks_right := TRUE;
IF stacker_crane_limit_right THEN
	stacker_crane_z_sp := 5.40;
END_IF	
END_IF  
//-----------------------------------------------------------------------------

// POSICION 33
IF GVL.POSICION = 33 AND count_forks=1 AND stacker_crane_limit_middle AND TIM_POSICION.Q  THEN
	  stacker_crane_x_sp := 6.45;
      stacker_crane_z_sp := 5.66;
END_IF 
// dejar carga posicion 33
IF GVL.POSICION = 33 AND TIM_POSICION.Q AND count_forks=1 AND gvl.x_position < 6.46 AND gvl.x_position > 6.44 AND gvl.Z_position < 5.67 AND gvl.Z_position > 5.65 THEN 
    Forks_right := TRUE;
IF stacker_crane_limit_right THEN
	stacker_crane_z_sp := 5.40;
END_IF	
END_IF  
//-----------------------------------------------------------------------------

// POSICION 34
IF GVL.POSICION = 34 AND count_forks=1 AND stacker_crane_limit_middle AND TIM_POSICION.Q  THEN
	  stacker_crane_x_sp := 7.51;
      stacker_crane_z_sp := 5.66;
END_IF 
// dejar carga posicion 34
IF GVL.POSICION = 34 AND TIM_POSICION.Q AND count_forks=1 AND gvl.x_position < 7.52 AND gvl.x_position > 7.50 AND gvl.Z_position < 5.67 AND gvl.Z_position > 5.65 THEN 
    Forks_right := TRUE;
IF stacker_crane_limit_right THEN
	stacker_crane_z_sp := 5.40;
END_IF	
END_IF  
//-----------------------------------------------------------------------------

// POSICION 35
IF GVL.POSICION = 35 AND count_forks=1 AND stacker_crane_limit_middle AND TIM_POSICION.Q  THEN
	  stacker_crane_x_sp := 8.59;
      stacker_crane_z_sp := 5.66;
END_IF 
// dejar carga posicion 35
IF GVL.POSICION = 35 AND TIM_POSICION.Q AND count_forks=1 AND gvl.x_position < 8.60 AND gvl.x_position > 8.58 AND gvl.Z_position < 5.67 AND gvl.Z_position > 5.65 THEN 
    Forks_right := TRUE;
IF stacker_crane_limit_right THEN
	stacker_crane_z_sp := 5.40;
END_IF	
END_IF  
//-----------------------------------------------------------------------------

// POSICION 36
IF GVL.POSICION = 36 AND count_forks=1 AND stacker_crane_limit_middle AND TIM_POSICION.Q  THEN
	  stacker_crane_x_sp := 9.66;
      stacker_crane_z_sp := 5.66;
END_IF 
// dejar carga posicion 36
IF GVL.POSICION = 36 AND TIM_POSICION.Q AND count_forks=1 AND gvl.x_position < 9.67 AND gvl.x_position > 9.65 AND gvl.Z_position < 5.67 AND gvl.Z_position > 5.65 THEN 
    Forks_right := TRUE;
IF stacker_crane_limit_right THEN
	stacker_crane_z_sp := 5.40;
END_IF	
END_IF 
//-----------------------------------------------------------------------------  

// --------- QUINTA FILA --------------

//-----------------------------------------------------------------------------
// POSICION 37
IF GVL.POSICION = 37 AND count_forks=1 AND stacker_crane_limit_middle AND TIM_POSICION.Q  THEN
	  stacker_crane_x_sp := 1.06;
      stacker_crane_z_sp := 7.50;
END_IF 
// dejar carga posicion 37
IF GVL.POSICION = 37 AND TIM_POSICION.Q AND count_forks=1 AND gvl.x_position < 1.07 AND gvl.x_position > 1.05 AND gvl.Z_position < 7.51 AND gvl.Z_position > 7.49 THEN 
    Forks_right := TRUE;
IF stacker_crane_limit_right THEN
	stacker_crane_z_sp := 7.30;
END_IF	
END_IF  
//-----------------------------------------------------------------------------

// POSICION 38
IF GVL.POSICION = 38 AND count_forks=1 AND stacker_crane_limit_middle AND TIM_POSICION.Q  THEN
	  stacker_crane_x_sp := 2.15;
      stacker_crane_z_sp := 7.50;
END_IF 
// dejar carga posicion 38
IF GVL.POSICION = 38 AND TIM_POSICION.Q AND count_forks=1 AND gvl.x_position < 2.16 AND gvl.x_position > 2.14 AND gvl.Z_position < 7.51 AND gvl.Z_position > 7.49 THEN 
    Forks_right := TRUE;
IF stacker_crane_limit_right THEN
	stacker_crane_z_sp := 7.30;
END_IF	
END_IF  
//-----------------------------------------------------------------------------

// POSICION 39
IF GVL.POSICION = 39 AND count_forks=1 AND stacker_crane_limit_middle AND TIM_POSICION.Q  THEN
	  stacker_crane_x_sp := 3.21;
      stacker_crane_z_sp := 7.50;
END_IF 
// dejar carga posicion 39
IF GVL.POSICION = 39 AND TIM_POSICION.Q AND count_forks=1 AND gvl.x_position < 3.22 AND gvl.x_position > 3.20 AND gvl.Z_position < 7.51 AND gvl.Z_position > 7.49 THEN 
    Forks_right := TRUE;
IF stacker_crane_limit_right THEN
	stacker_crane_z_sp := 7.30;
END_IF	
END_IF  
//-----------------------------------------------------------------------------

// POSICION 40
IF GVL.POSICION = 40 AND count_forks=1 AND stacker_crane_limit_middle AND TIM_POSICION.Q  THEN
	  stacker_crane_x_sp := 4.29;
      stacker_crane_z_sp := 7.50;
END_IF 
// dejar carga posicion 40
IF GVL.POSICION = 40 AND TIM_POSICION.Q AND count_forks=1 AND gvl.x_position < 4.30 AND gvl.x_position > 4.28 AND gvl.Z_position < 7.51 AND gvl.Z_position > 7.49 THEN 
    Forks_right := TRUE;
IF stacker_crane_limit_right THEN
	stacker_crane_z_sp := 7.30;
END_IF	
END_IF  
//-----------------------------------------------------------------------------

// POSICION 41
IF GVL.POSICION = 41 AND count_forks=1 AND stacker_crane_limit_middle AND TIM_POSICION.Q  THEN
	  stacker_crane_x_sp := 5.36;
      stacker_crane_z_sp := 7.50;
END_IF 
// dejar carga posicion 41
IF GVL.POSICION = 41 AND TIM_POSICION.Q AND count_forks=1 AND gvl.x_position < 5.37 AND gvl.x_position > 5.35 AND gvl.Z_position < 7.51 AND gvl.Z_position > 7.49 THEN 
    Forks_right := TRUE;
IF stacker_crane_limit_right THEN
	stacker_crane_z_sp := 7.30;
END_IF	
END_IF  
//-----------------------------------------------------------------------------

// POSICION 42
IF GVL.POSICION = 42 AND count_forks=1 AND stacker_crane_limit_middle AND TIM_POSICION.Q  THEN
	  stacker_crane_x_sp := 6.45;
      stacker_crane_z_sp := 7.50;
END_IF 
// dejar carga posicion 42
IF GVL.POSICION = 42 AND TIM_POSICION.Q AND count_forks=1 AND gvl.x_position < 6.46 AND gvl.x_position > 6.44 AND gvl.Z_position < 7.51 AND gvl.Z_position > 7.49 THEN 
    Forks_right := TRUE;
IF stacker_crane_limit_right THEN
	stacker_crane_z_sp := 7.30;
END_IF	
END_IF  
//-----------------------------------------------------------------------------

// POSICION 43
IF GVL.POSICION = 43 AND count_forks=1 AND stacker_crane_limit_middle AND TIM_POSICION.Q  THEN
	  stacker_crane_x_sp := 7.51;
      stacker_crane_z_sp := 7.50;
END_IF 
// dejar carga posicion 43
IF GVL.POSICION = 43 AND TIM_POSICION.Q AND count_forks=1 AND gvl.x_position < 7.52 AND gvl.x_position > 7.50 AND gvl.Z_position < 7.51 AND gvl.Z_position > 7.49 THEN 
    Forks_right := TRUE;
IF stacker_crane_limit_right THEN
	stacker_crane_z_sp := 7.30;
END_IF	
END_IF  
//-----------------------------------------------------------------------------

// POSICION 44
IF GVL.POSICION = 44 AND count_forks=1 AND stacker_crane_limit_middle AND TIM_POSICION.Q  THEN
	  stacker_crane_x_sp := 8.59;
      stacker_crane_z_sp := 7.50;
END_IF 
// dejar carga posicion 44
IF GVL.POSICION = 44 AND TIM_POSICION.Q AND count_forks=1 AND gvl.x_position < 8.60 AND gvl.x_position > 8.58 AND gvl.Z_position < 7.51 AND gvl.Z_position > 7.49 THEN 
    Forks_right := TRUE;
IF stacker_crane_limit_right THEN
	stacker_crane_z_sp := 7.30;
END_IF	
END_IF  
//-----------------------------------------------------------------------------

// POSICION 45
IF GVL.POSICION = 45 AND count_forks=1 AND stacker_crane_limit_middle AND TIM_POSICION.Q  THEN
	  stacker_crane_x_sp := 9.66;
      stacker_crane_z_sp := 7.50;
END_IF 
// dejar carga posicion 45
IF GVL.POSICION = 45 AND TIM_POSICION.Q AND count_forks=1 AND gvl.x_position < 9.67 AND gvl.x_position > 9.65 AND gvl.Z_position < 7.51 AND gvl.Z_position > 7.49 THEN 
    Forks_right := TRUE;
IF stacker_crane_limit_right THEN
	stacker_crane_z_sp := 7.30;
END_IF	
END_IF 
//----------------------------------------------------------------------------- 

// --------- SEXTA FILA --------------

//-----------------------------------------------------------------------------
// POSICION 46
IF GVL.POSICION = 46 AND count_forks=1 AND stacker_crane_limit_middle AND TIM_POSICION.Q  THEN
	  stacker_crane_x_sp := 1.06;
      stacker_crane_z_sp := 9.20;
END_IF 
// dejar carga posicion 46
IF GVL.POSICION = 46 AND TIM_POSICION.Q AND count_forks=1 AND gvl.x_position < 1.07 AND gvl.x_position > 1.05 AND gvl.Z_position < 9.21 AND gvl.Z_position > 9.19 THEN 
    Forks_right := TRUE;
IF stacker_crane_limit_right THEN
	stacker_crane_z_sp := 9.0;
END_IF	
END_IF  
//-----------------------------------------------------------------------------

// POSICION 47
IF GVL.POSICION = 47 AND count_forks=1 AND stacker_crane_limit_middle AND TIM_POSICION.Q  THEN
	  stacker_crane_x_sp := 2.15;
      stacker_crane_z_sp := 9.20;
END_IF 
// dejar carga posicion 47
IF GVL.POSICION = 47 AND TIM_POSICION.Q AND count_forks=1 AND gvl.x_position < 2.16 AND gvl.x_position > 2.14 AND gvl.Z_position < 9.21 AND gvl.Z_position > 9.19 THEN 
    Forks_right := TRUE;
IF stacker_crane_limit_right THEN
	stacker_crane_z_sp := 9.0;
END_IF	
END_IF  
//-----------------------------------------------------------------------------

// POSICION 48
IF GVL.POSICION = 48 AND count_forks=1 AND stacker_crane_limit_middle AND TIM_POSICION.Q  THEN
	  stacker_crane_x_sp := 3.21;
      stacker_crane_z_sp := 9.20;
END_IF 
// dejar carga posicion 48
IF GVL.POSICION = 48 AND TIM_POSICION.Q AND count_forks=1 AND gvl.x_position < 3.22 AND gvl.x_position > 3.20 AND gvl.Z_position < 9.21 AND gvl.Z_position > 9.19 THEN 
    Forks_right := TRUE;
IF stacker_crane_limit_right THEN
	stacker_crane_z_sp := 9.0;
END_IF	
END_IF  
//-----------------------------------------------------------------------------

// POSICION 49
IF GVL.POSICION = 49 AND count_forks=1 AND stacker_crane_limit_middle AND TIM_POSICION.Q  THEN
	  stacker_crane_x_sp := 4.29;
      stacker_crane_z_sp := 9.20;
END_IF 
// dejar carga posicion 49
IF GVL.POSICION = 49 AND TIM_POSICION.Q AND count_forks=1 AND gvl.x_position < 4.30 AND gvl.x_position > 4.28 AND gvl.Z_position < 9.21 AND gvl.Z_position > 9.19 THEN 
    Forks_right := TRUE;
IF stacker_crane_limit_right THEN
	stacker_crane_z_sp := 9.0;
END_IF	
END_IF  
//-----------------------------------------------------------------------------

// POSICION 50
IF GVL.POSICION = 50 AND count_forks=1 AND stacker_crane_limit_middle AND TIM_POSICION.Q  THEN
	  stacker_crane_x_sp := 5.36;
      stacker_crane_z_sp := 9.20;
END_IF 
// dejar carga posicion 50
IF GVL.POSICION = 50 AND TIM_POSICION.Q AND count_forks=1 AND gvl.x_position < 5.37 AND gvl.x_position > 5.35 AND gvl.Z_position < 9.21 AND gvl.Z_position > 9.19 THEN 
    Forks_right := TRUE;
IF stacker_crane_limit_right THEN
	stacker_crane_z_sp := 9.0;
END_IF	
END_IF  
//-----------------------------------------------------------------------------

// POSICION 51
IF GVL.POSICION = 51 AND count_forks=1 AND stacker_crane_limit_middle AND TIM_POSICION.Q  THEN
	  stacker_crane_x_sp := 6.45;
      stacker_crane_z_sp := 9.20;
END_IF 
// dejar carga posicion 51
IF GVL.POSICION = 51 AND TIM_POSICION.Q AND count_forks=1 AND gvl.x_position < 6.46 AND gvl.x_position > 6.44 AND gvl.Z_position < 9.21 AND gvl.Z_position > 9.19 THEN 
    Forks_right := TRUE;
IF stacker_crane_limit_right THEN
	stacker_crane_z_sp := 9.0;
END_IF	
END_IF  
//-----------------------------------------------------------------------------

// POSICION 52
IF GVL.POSICION = 52 AND count_forks=1 AND stacker_crane_limit_middle AND TIM_POSICION.Q  THEN
	  stacker_crane_x_sp := 7.51;
      stacker_crane_z_sp := 9.20;
END_IF 
// dejar carga posicion 52
IF GVL.POSICION = 52 AND TIM_POSICION.Q AND count_forks=1 AND gvl.x_position < 7.52 AND gvl.x_position > 7.50 AND gvl.Z_position < 9.21 AND gvl.Z_position > 9.19 THEN 
    Forks_right := TRUE;
IF stacker_crane_limit_right THEN
	stacker_crane_z_sp := 9.0;
END_IF	
END_IF  
//-----------------------------------------------------------------------------

// POSICION 53
IF GVL.POSICION = 53 AND count_forks=1 AND stacker_crane_limit_middle AND TIM_POSICION.Q  THEN
	  stacker_crane_x_sp := 8.59;
      stacker_crane_z_sp := 9.20;
END_IF 
// dejar carga posicion 53
IF GVL.POSICION = 53 AND TIM_POSICION.Q AND count_forks=1 AND gvl.x_position < 8.60 AND gvl.x_position > 8.58 AND gvl.Z_position < 9.21 AND gvl.Z_position > 9.19 THEN 
    Forks_right := TRUE;
IF stacker_crane_limit_right THEN
	stacker_crane_z_sp := 9.0;
END_IF	
END_IF  
//-----------------------------------------------------------------------------

// POSICION 54
IF GVL.POSICION = 54 AND count_forks=1 AND stacker_crane_limit_middle AND TIM_POSICION.Q  THEN
	  stacker_crane_x_sp := 9.66;
      stacker_crane_z_sp := 9.20;
END_IF 
// dejar carga posicion 54
IF GVL.POSICION = 54 AND TIM_POSICION.Q AND count_forks=1 AND gvl.x_position < 9.67 AND gvl.x_position > 9.65 AND gvl.Z_position < 9.21 AND gvl.Z_position > 9.19 THEN 
    Forks_right := TRUE;
IF stacker_crane_limit_right THEN
	stacker_crane_z_sp := 9.0;
END_IF	
END_IF 
//----------------------------------------------------------------------------- 


//---------------- RECOGER UÑA Y VOLVER A INICIO----------------------------------- 



//-----------------------------------------------------------------------------
	// RETARDO RECOGIDA UÑAS ABAJO
    Tim_descarga(IN := stacker_crane_limit_right AND stacker_crane_z_sp < 0.41 AND stacker_crane_z_sp > 0.39 , PT:= T#1S);
IF Tim_descarga.Q	THEN
	Forks_right := FALSE;
	count_forks := 0;
END_IF	
IF MANDAR_POSICION AND TIM_DESCARGA.Q THEN
	RESET_NUMERO_ESTANTE := TRUE;
END_IF

	// RETARDO RECOGIDA UÑAS SEGUNDA ALTURA
    Tim_descarga1(IN := stacker_crane_limit_right AND stacker_crane_z_sp < 2.01 AND stacker_crane_z_sp > 1.99 , PT:= T#1S);
IF Tim_descarga1.Q	THEN
	Forks_right := FALSE;
	count_forks := 0;
END_IF
IF MANDAR_POSICION AND TIM_DESCARGA1.Q THEN
	RESET_NUMERO_ESTANTE := TRUE;
END_IF

	// RETARDO RECOGIDA UÑAS TERCERA ALTURA
    Tim_descarga2(IN := stacker_crane_limit_right AND stacker_crane_z_sp < 3.91 AND stacker_crane_z_sp > 3.89, PT:= T#1S);
IF Tim_descarga2.Q	THEN
	Forks_right := FALSE;
	count_forks := 0;
END_IF
IF MANDAR_POSICION AND TIM_DESCARGA2.Q THEN
	RESET_NUMERO_ESTANTE := TRUE;
END_IF

	// RETARDO RECOGIDA UÑAS CUARTA ALTURA
    Tim_descarga3(IN := stacker_crane_limit_right AND stacker_crane_z_sp < 5.41 AND stacker_crane_z_sp > 5.39, PT:= T#1S);
IF Tim_descarga3.Q	THEN
	Forks_right := FALSE;
	count_forks := 0;
END_IF
IF MANDAR_POSICION AND TIM_DESCARGA3.Q THEN
	RESET_NUMERO_ESTANTE := TRUE;
END_IF

    // RETARDO RECOGIDA UÑAS QUINTA ALTURA
    Tim_descarga4(IN := stacker_crane_limit_right AND stacker_crane_z_sp < 7.31 AND stacker_crane_z_sp > 7.29, PT:= T#1S);
IF Tim_descarga4.Q	THEN
	Forks_right := FALSE;
	count_forks := 0;
END_IF
IF MANDAR_POSICION AND TIM_DESCARGA4.Q THEN
	RESET_NUMERO_ESTANTE := TRUE;
END_IF

    // RETARDO RECOGIDA UÑAS SEXTA ALTURA
    Tim_descarga5(IN := stacker_crane_limit_right AND stacker_crane_z_sp < 9.01 AND stacker_crane_z_sp > 8.99, PT:= T#1S);
IF Tim_descarga5.Q	THEN
	Forks_right := FALSE;
	count_forks := 0;
END_IF
IF MANDAR_POSICION AND TIM_DESCARGA5.Q THEN
	RESET_NUMERO_ESTANTE := TRUE;
END_IF

// VUELTA DESDE UBICACION DE DESCARGA EN ESTANTERIA A UBICACION DE CARGA
IF NOT FORKS_RIGHT AND COUNT_FORKS =0 AND stacker_crane_limit_middle AND TRASLO_CARGADO THEN
	TRASLO_CARGADO := FALSE;
    stacker_crane_x_sp := 0;
    stacker_crane_Z_sp := 0;
	CTU_MOV.RESET := FALSE;
END_IF

//-------- VISUALIZACION UBICACION EN INSTRUMENTACION DEL CUADRO-------------
  GVL.NUMERO_ESTANTE := CTU_MOV.CV;
  
//-------- ocupacion de estanterias color azul-----------
STARTFP(CLK:= flanco_forks_out );

IF gvl.POSICION = 1 AND startfp.Q THEN
pos1:= 1; 
pos := POS + 1;
REGISTRO[POS] := 1;
END_IF
IF gvl.POSICION = 2 AND startfp.Q THEN
pos2:= 1;
POS := POS + 1;
REGISTRO[POS] := 2;
END_IF
IF gvl.POSICION = 3 AND startfp.Q THEN 
pos3:= 1;
POS := POS + 1;
REGISTRO[POS] := 3;
END_IF
IF gvl.POSICION = 4 AND startfp.Q THEN
pos4:= 1;
pos := POS + 1;
REGISTRO[POS] := 4;
END_IF
IF gvl.POSICION = 5 AND startfp.Q THEN
pos5:= 1;
pos := POS + 1;
REGISTRO[POS] := 5;
END_IF
IF gvl.POSICION = 6 AND startfp.Q THEN
pos6:= 1;
pos := POS + 1;
REGISTRO[POS] := 6;
END_IF
IF gvl.POSICION = 7 AND startfp.Q THEN
pos7:= 1;
pos := POS + 1;
REGISTRO[POS] := 7;
END_IF
IF gvl.POSICION = 8 AND startfp.Q THEN
pos8:= 1;
pos := POS + 1;
REGISTRO[POS] := 8;
END_IF
IF gvl.POSICION = 9 AND startfp.Q THEN
pos9:= 1;
pos := POS + 1;
REGISTRO[POS] := 9;
END_IF
IF gvl.POSICION = 10 AND startfp.Q THEN
pos10:= 1;
pos := POS + 1;
REGISTRO[POS] := 10;
END_IF
IF gvl.POSICION = 11 AND startfp.Q THEN
pos11:= 1;
pos := POS + 1;
REGISTRO[POS] := 11;
END_IF
IF gvl.POSICION = 12 AND startfp.Q THEN
pos12:= 1;
pos := POS + 1;
REGISTRO[POS] := 12;
END_IF
IF gvl.POSICION = 13 AND startfp.Q THEN 
pos13:= 1;
pos := POS + 1;
REGISTRO[POS] := 13;
END_IF
IF gvl.POSICION = 14 AND startfp.Q THEN
pos14:= 1;
pos := POS + 1;
REGISTRO[POS] := 14;
END_IF
IF gvl.POSICION = 15 AND startfp.Q THEN
pos15:= 1;
pos := POS + 1;
REGISTRO[POS] := 15;
END_IF
IF gvl.POSICION = 16 AND startfp.Q THEN
pos16:= 1;
pos := POS + 1;
REGISTRO[POS] := 16;
END_IF
IF gvl.POSICION = 17 AND startfp.Q THEN
pos17:= 1;
pos := POS + 1;
REGISTRO[POS] := 17;
END_IF
IF gvl.POSICION = 18 AND startfp.Q THEN
pos18:= 1; 
pos := POS + 1;
REGISTRO[POS] := 18;
END_IF

//-------- ocupacion de estanterias color verde-----------
IF gvl.POSICION = 19 AND startfp.Q THEN
pos19:= 1;
pos := POS + 1;
REGISTRO[POS] := 19;
END_IF
IF gvl.POSICION = 20 AND startfp.Q THEN
pos20:= 1;
pos := POS + 1;
REGISTRO[POS] := 20;
END_IF
IF gvl.POSICION = 21 AND startfp.Q THEN
pos21:= 1;
pos := POS + 1;
REGISTRO[POS] := 21;
END_IF
IF gvl.POSICION = 22 AND startfp.Q THEN
pos22:= 1;
pos := POS + 1;
REGISTRO[POS] := 22;
END_IF
IF gvl.POSICION = 23 AND startfp.Q THEN
pos23:= 1;
pos := POS + 1;
REGISTRO[POS] := 23;
END_IF
IF gvl.POSICION = 24 AND startfp.Q THEN
pos24:= 1;
pos := POS + 1;
REGISTRO[POS] := 24;
END_IF
IF gvl.POSICION = 25 AND startfp.Q THEN
pos25:= 1;
pos := POS + 1;
REGISTRO[POS] := 25;
END_IF
IF gvl.POSICION = 26 AND startfp.Q THEN
pos26:= 1;
pos := POS + 1;
REGISTRO[POS] := 26;
END_IF
IF gvl.POSICION = 27 AND startfp.Q THEN
pos27:= 1;
pos := POS + 1;
REGISTRO[POS] := 27;
END_IF
IF gvl.POSICION = 28 AND startfp.Q THEN
pos28:= 1;
pos := POS + 1;
REGISTRO[POS] := 28;
END_IF
IF gvl.POSICION = 29 AND startfp.Q THEN
pos29:= 1;
pos := POS + 1;
REGISTRO[POS] := 29;
END_IF
IF gvl.POSICION = 30 AND startfp.Q THEN
pos30:= 1;
pos := POS + 1;
REGISTRO[POS] := 30;
END_IF
IF gvl.POSICION = 31 AND startfp.Q THEN
pos31:= 1;
pos := POS + 1;
REGISTRO[POS] := 31;
END_IF
IF gvl.POSICION = 32 AND startfp.Q THEN
pos32:= 1;
pos := POS + 1;
REGISTRO[POS] := 32;
END_IF
IF gvl.POSICION = 33 AND startfp.Q THEN
pos33:= 1;
pos := POS + 1;
REGISTRO[POS] := 33;
END_IF
IF gvl.POSICION = 34 AND startfp.Q THEN
pos34:= 1;
pos := POS + 1;
REGISTRO[POS] := 34;
END_IF
IF gvl.POSICION = 35 AND startfp.Q THEN
pos35:= 1;
pos := POS + 1;
REGISTRO[POS] := 35;
END_IF
IF gvl.POSICION = 36 AND startfp.Q THEN
pos36:= 1;
pos := POS + 1;
REGISTRO[POS] := 36;
END_IF

//-------- ocupacion de estanterias color metal-----------
IF gvl.POSICION = 37 AND startfp.Q THEN
pos37:= 1;
pos := POS + 1;
REGISTRO[POS] := 37;
END_IF
IF gvl.POSICION = 38 AND startfp.Q THEN
pos38:= 1;
pos := POS + 1;
REGISTRO[POS] := 38;
END_IF
IF gvl.POSICION = 39 AND startfp.Q THEN
pos39:= 1;
pos := POS + 1;
REGISTRO[POS] := 39;
END_IF
IF gvl.POSICION = 40 AND startfp.Q THEN
pos40:= 1;
pos := POS + 1;
REGISTRO[POS] := 40;
END_IF
IF gvl.POSICION = 41 AND startfp.Q THEN
pos41:= 1;
pos := POS + 1;
REGISTRO[POS] := 41;
END_IF
IF gvl.POSICION = 42 AND startfp.Q THEN
pos42:= 1;
pos := POS + 1;
REGISTRO[POS] := 42;
END_IF
IF gvl.POSICION = 43 AND startfp.Q THEN
pos43:= 1;
pos := POS + 1;
REGISTRO[POS] := 43;
END_IF
IF gvl.POSICION = 44 AND startfp.Q THEN
pos44:= 1;
pos := POS + 1;
REGISTRO[POS] := 44;
END_IF
IF gvl.POSICION = 45 AND startfp.Q THEN
pos45:= 1;
pos := POS + 1;
REGISTRO[POS] := 45;
END_IF
IF gvl.POSICION = 46 AND startfp.Q THEN
pos46:= 1;
pos := POS + 1;
REGISTRO[POS] := 46;
END_IF
IF gvl.POSICION = 47 AND startfp.Q THEN
pos47:= 1;
pos := POS + 1;
REGISTRO[POS] := 47;
END_IF
IF gvl.POSICION = 48 AND startfp.Q THEN
pos48:= 1;
pos := POS + 1;
REGISTRO[POS] := 48;
END_IF
IF gvl.POSICION = 49 AND startfp.Q THEN
pos49:= 1;
pos := POS + 1;
REGISTRO[POS] := 49;
END_IF
IF gvl.POSICION = 50 AND startfp.Q THEN
pos50:= 1;
pos := POS + 1;
REGISTRO[POS] := 50;
END_IF
IF gvl.POSICION = 51 AND startfp.Q THEN
pos51:= 1;
pos := POS + 1;
REGISTRO[POS] := 51;
END_IF
IF gvl.POSICION = 52 AND startfp.Q THEN
pos52:= 1;
pos := POS + 1;
REGISTRO[POS] := 52;
END_IF
IF gvl.POSICION = 53 AND startfp.Q THEN
pos53:= 1;
pos := POS + 1;
REGISTRO[POS] := 53;
END_IF
IF gvl.POSICION = 54 AND startfp.Q THEN
pos54:= 1;
pos := POS + 1;
REGISTRO[POS] := 54;
END_IF

//------- saturacion color azul-------
IF pos1 AND pos2 AND pos3 AND pos4 AND pos5 AND pos6 AND pos7 AND pos7 AND pos8 AND pos9 AND pos10 AND pos11 AND pos12 AND pos13 AND pos14 AND pos15 AND pos16 AND pos17 AND pos18
	THEN color_azul_saturado := 1;
END_IF
//------- saturacion color verde-------
IF pos19 AND pos20 AND pos21 AND pos22 AND pos23 AND pos24 AND pos25 AND pos26 AND pos27 AND pos28 AND pos29 AND pos30 AND pos31 AND pos32 AND pos33 AND pos34 AND pos35 AND pos36 
	THEN color_verde_saturado := 1;
END_IF
//------- saturacion color metal-------
IF pos37 AND pos38 AND pos39 AND pos40 AND pos41 AND pos42 AND pos43 AND pos44 AND pos45 AND pos46 AND pos47 AND pos48 AND pos49 AND pos50 AND pos51 AND pos52 AND pos53 AND pos54 
	THEN color_metal_saturado := 1;
END_IF
IF reset and color_azul_saturado OR color_verde_saturado OR color_metal_saturado THEN
	color_azul_saturado := 0;
	color_verde_saturado := 0;
	color_metal_saturado := 0;
END_IF
//----------- ALARMA POR SATURACION ------------
IF color_azul_saturado OR color_verde_saturado OR color_metal_saturado OR CNT_TOTAL.Q THEN ALARMA_ACTIVA := 1;
END_IF
IF NOT color_azul_saturado AND NOT color_verde_saturado AND NOT color_metal_saturado AND NOT CNT_TOTAL.Q THEN ALARMA_ACTIVA := 0;
END_IF
IF ALARMA_ACTIVA THEN
	Emisor_piezas := FALSE;
	cinta_piezas := FALSE;
	Emisor_piezas := FALSE;
END_IF
//----------------- ROBOT ARTICULADO -----------------------

// emisor piezas a robot
IF SYS_ON AND NOT ALARMA_ACTIVA THEN
	Emisor_piezas := TRUE;
END_IF
IF Emisor_piezas AND NOT SYS_ON OR FALLO_ROBOT OR ALARMA_ACTIVA THEN
	Emisor_piezas := FALSE;
END_IF

// cinta piezas robot
IF SYS_ON AND NOT robot_ocupado AND NOT ALARMA_ACTIVA THEN
	cinta_piezas := TRUE;
END_IF
IF cinta_piezas AND SENSOR_piezas_cinta AND robot_ocupado OR NOT SYS_ON THEN
	cinta_piezas := FALSE;
END_IF

// MARCHA ROBOT
IF SYS_ON AND NOT robot_ocupado THEN 
	ON_ROBOT := TRUE;
END_IF
IF NOT SYS_ON THEN 
	ON_ROBOT := FALSE;
END_IF

//------------------ ROBOT CARTESIANO ---------------------
IF NOT sys_on THEN
	bajar_robot_cartesiano := FALSE ;
	agarrar_pieza_robot_cart := FALSE ;
	avanzar_robot_cartesiano := FALSE ;
	fin_ciclo_robot_cartesiano := FALSE ;
	bit1 := 0 ;
	END_IF
// CINTA PIEZAS ACABADAS Y TOPE	
IF SYS_ON AND NOT ALARMA_ACTIVA THEN
CINTA_PIEZAS_ACABADAS := TRUE ;
TOPE_PIEZAS := TRUE ;
ELSE 	
CINTA_PIEZAS_ACABADAS := FALSE ;
TOPE_PIEZAS := FALSE ;	
END_IF
// bajar
IF sys_on AND detec_piezas_cartesiano AND NOT SENSOR_0 THEN
	bajar_robot_cartesiano := TRUE ;
	bit1 := 1;
END_IF
// coger pieza
TON_bajar1 (IN:=sys_on AND bit1 = 1 AND detec_piezas_cartesiano, PT:= T#1S);
IF sys_on AND TON_bajar1.Q AND deteccion_pieza_robot_cart THEN
	agarrar_pieza_robot_cart := TRUE ;
	bit1 := 2;
// subir	
END_IF
IF sys_on AND bit1 = 2 THEN 
	bajar_robot_cartesiano := FALSE ;
	bit1 := 3;
END_IF	
// avanzar
TON_subir1 (IN:=sys_on AND bit1 = 3, PT:= T#1S);
IF sys_on AND TON_subir1.Q THEN 
	avanzar_robot_cartesiano := TRUE ;
	bit1 := 4;
END_IF	
// bajar 2
TON_avanzar (IN:=sys_on AND bit1 = 4 AND agarrar_pieza_robot_cart, PT:= T#1S);
IF sys_on AND TON_avanzar.Q THEN 
	bajar_robot_cartesiano := TRUE ;
	bit1 := 5;
END_IF	
// dejar pieza	
TON_bajar2 (IN:=sys_on AND bit1 = 5 AND agarrar_pieza_robot_cart, PT:= T#1S);
IF sys_on AND TON_bajar2.Q THEN 	
	agarrar_pieza_robot_cart := FALSE ;
	bit1 := 6;
END_IF
// subir 2	
IF sys_on AND NOT agarrar_pieza_robot_cart AND bit1 = 6 THEN 	
	bajar_robot_cartesiano := FALSE ;
	bit1 := 7;
END_IF
// recoger brazo
TON_subir2 (IN:=sys_on AND bit1 = 7 AND NOT agarrar_pieza_robot_cart AND NOT fin_ciclo_robot_cartesiano, PT:= T#1S);
IF sys_on AND TON_subir2.Q THEN 	
	avanzar_robot_cartesiano := FALSE ;	
	bit1 := 8;
END_IF	
// fin ciclo
TON_retroceder (IN:= sys_on AND NOT avanzar_robot_cartesiano AND bit1 = 8, PT:= T#1S);
IF sys_on AND TON_retroceder.Q THEN 	
	fin_ciclo_robot_cartesiano := TRUE ;
	bit1 := 9;
END_IF	
// reset fin ciclo
TON_reset(IN:= sys_on  AND bit1 = 9 , PT:= T#1S);
IF TON_reset.Q THEN 	
	fin_ciclo_robot_cartesiano := FALSE ;
	bit1 := 10;
END_IF

END_PROGRAM

// Device/Application/ANALOGICAS
PROGRAM ANALOGICAS
VAR
	ESCALADO_X: ESCALADO;
	ESCALADO_Z: ESCALADO;
END_VAR

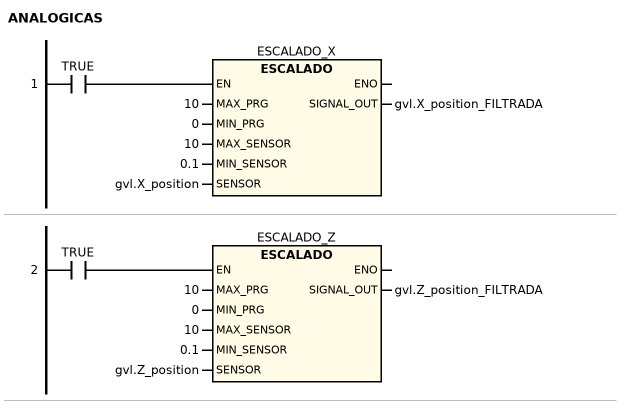
// NETWORK 1
ESCALADO_X(
    MAX_PRG := 10,
    MIN_PRG := 0,
    MAX_SENSOR := 10,
    MIN_SENSOR := 0.1,
    SENSOR := gvl.X_position,
    SIGNAL_OUT => gvl.X_position_FILTRADA); // ESCALADO

// NETWORK 2
ESCALADO_Z(
    MAX_PRG := 10,
    MIN_PRG := 0,
    MAX_SENSOR := 10,
    MIN_SENSOR := 0.1,
    SENSOR := gvl.Z_position,
    SIGNAL_OUT => gvl.Z_position_FILTRADA); // ESCALADO

END_PROGRAM

// Device/Application/ESCALADO
FUNCTION_BLOCK ESCALADO
VAR_INPUT
	MAX_PRG: REAL;
	MIN_PRG: REAL;
	MAX_SENSOR: REAL;
	MIN_SENSOR: REAL;
	SENSOR: REAL;
END_VAR
VAR_OUTPUT
	SIGNAL_OUT: REAL;
END_VAR
VAR
END_VAR

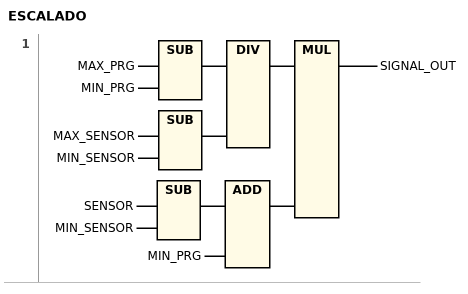
// NETWORK 1
SIGNAL_OUT := ((MAX_PRG - MIN_PRG) / (MAX_SENSOR - MIN_SENSOR)) * ((SENSOR - MIN_SENSOR) + MIN_PRG);

END_FUNCTION_BLOCK

// Device/Application/Panel_control
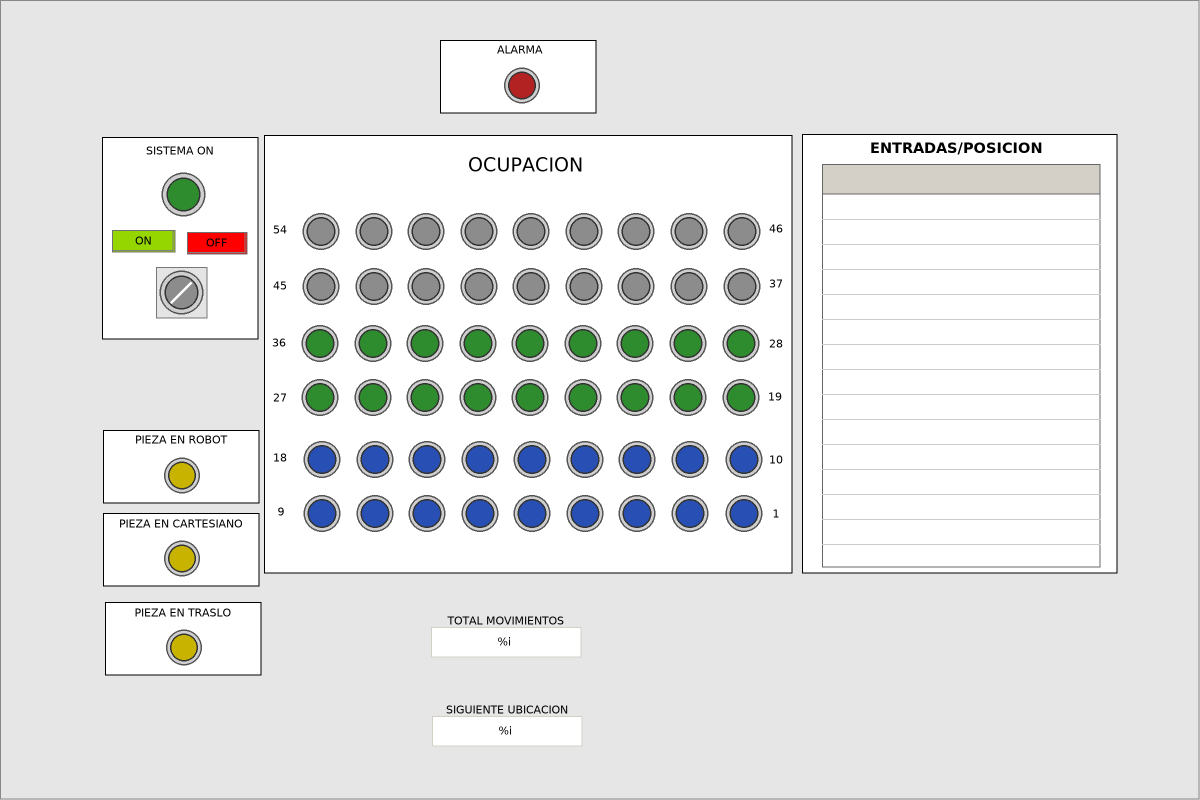
VISUALIZATION Panel_control  // 1200x800
    Rectangle (440,40 156x73)
    Rectangle (802,134 315x439)
    Rectangle (103,513 156x73)
    Rectangle (102,137 156x202)
    Button (112,230 63x22), "ON"
        tap PLC_PRG.Start
    Lamp1 (155,169 57x51), variable: PLC_PRG.sys_on, style: Lamp-Lamp1-Green
    Button (187,232 60x22), "OFF"
        tap PLC_PRG.Stop
    RotarySwitch (153,267 57x51), variable: PLC_PRG.auto, behaviour: TOGGLE, style: Switch-RotarySwitch-Gray
    Rectangle (264,135 528x438)
    Lamp1 (664,322 48x43), variable: PLC_PRG.pos29, style: Lamp-Lamp1-Green
    Lamp1 (611,322 48x43), variable: PLC_PRG.pos30, style: Lamp-Lamp1-Green
    Lamp1 (559,322 48x43), variable: PLC_PRG.pos31, style: Lamp-Lamp1-Green
    Lamp1 (506,322 48x43), variable: PLC_PRG.pos32, style: Lamp-Lamp1-Green
    Lamp1 (454,322 48x43), variable: PLC_PRG.pos33, style: Lamp-Lamp1-Green
    Lamp1 (401,322 48x43), variable: PLC_PRG.pos34, style: Lamp-Lamp1-Green
    Lamp1 (717,322 48x43), variable: PLC_PRG.pos28, style: Lamp-Lamp1-Green
    Lamp1 (349,322 48x43), variable: PLC_PRG.pos35, style: Lamp-Lamp1-Green
    Lamp1 (296,322 48x43), variable: PLC_PRG.pos36, style: Lamp-Lamp1-Green
    Lamp1 (664,376 48x43), variable: PLC_PRG.pos20, style: Lamp-Lamp1-Green
    Lamp1 (611,376 48x43), variable: PLC_PRG.pos21, style: Lamp-Lamp1-Green
    Lamp1 (559,376 48x43), variable: PLC_PRG.pos22, style: Lamp-Lamp1-Green
    Lamp1 (506,376 48x43), variable: PLC_PRG.pos23, style: Lamp-Lamp1-Green
    Lamp1 (454,376 48x43), variable: PLC_PRG.pos24, style: Lamp-Lamp1-Green
    Lamp1 (401,376 48x43), variable: PLC_PRG.pos25, style: Lamp-Lamp1-Green
    Lamp1 (717,376 48x43), variable: PLC_PRG.pos19, style: Lamp-Lamp1-Green
    Lamp1 (349,376 48x43), variable: PLC_PRG.pos26, style: Lamp-Lamp1-Green
    Lamp1 (296,376 48x43), variable: PLC_PRG.pos27, style: Lamp-Lamp1-Green
    Lamp1 (665,210 48x43), variable: PLC_PRG.pos47, style: Lamp-Lamp1-Gray
    Lamp1 (612,210 48x43), variable: PLC_PRG.pos48, style: Lamp-Lamp1-Gray
    Lamp1 (560,210 48x43), variable: PLC_PRG.pos49, style: Lamp-Lamp1-Gray
    Lamp1 (507,210 48x43), variable: PLC_PRG.pos50, style: Lamp-Lamp1-Gray
    Lamp1 (455,210 48x43), variable: PLC_PRG.pos51, style: Lamp-Lamp1-Gray
    Lamp1 (402,210 48x43), variable: PLC_PRG.pos52, style: Lamp-Lamp1-Gray
    Lamp1 (718,210 48x43), variable: PLC_PRG.pos46, style: Lamp-Lamp1-Gray
    Lamp1 (350,210 48x43), variable: PLC_PRG.pos53, style: Lamp-Lamp1-Gray
    Lamp1 (297,210 48x43), variable: PLC_PRG.pos54, style: Lamp-Lamp1-Gray
    Lamp1 (665,265 48x43), variable: PLC_PRG.pos38, style: Lamp-Lamp1-Gray
    Lamp1 (612,265 48x43), variable: PLC_PRG.pos39, style: Lamp-Lamp1-Gray
    Lamp1 (560,265 48x43), variable: PLC_PRG.pos40, style: Lamp-Lamp1-Gray
    Lamp1 (507,265 48x43), variable: PLC_PRG.pos41, style: Lamp-Lamp1-Gray
    Lamp1 (455,265 48x43), variable: PLC_PRG.pos42, style: Lamp-Lamp1-Gray
    Lamp1 (402,265 48x43), variable: PLC_PRG.pos43, style: Lamp-Lamp1-Gray
    Lamp1 (718,265 48x43), variable: PLC_PRG.pos37, style: Lamp-Lamp1-Gray
    Lamp1 (350,265 48x43), variable: PLC_PRG.pos44, style: Lamp-Lamp1-Gray
    Lamp1 (297,265 48x43), variable: PLC_PRG.pos45, style: Lamp-Lamp1-Gray
    Lamp1 (666,438 48x43), variable: PLC_PRG.pos11, style: Lamp-Lamp1-Blue
    Lamp1 (613,438 48x43), variable: PLC_PRG.pos12, style: Lamp-Lamp1-Blue
    Lamp1 (561,438 48x43), variable: PLC_PRG.pos13, style: Lamp-Lamp1-Blue
    Lamp1 (508,438 48x43), variable: PLC_PRG.pos14, style: Lamp-Lamp1-Blue
    Lamp1 (456,438 48x43), variable: PLC_PRG.pos15, style: Lamp-Lamp1-Blue
    Lamp1 (403,438 48x43), variable: PLC_PRG.pos16, style: Lamp-Lamp1-Blue
    Lamp1 (720,438 48x43), variable: PLC_PRG.pos10, style: Lamp-Lamp1-Blue
    Lamp1 (351,438 48x43), variable: PLC_PRG.pos17, style: Lamp-Lamp1-Blue
    Lamp1 (298,438 48x43), variable: PLC_PRG.pos18, style: Lamp-Lamp1-Blue
    Lamp1 (666,492 48x43), variable: PLC_PRG.pos2, style: Lamp-Lamp1-Blue
    Lamp1 (613,492 48x43), variable: PLC_PRG.pos3, style: Lamp-Lamp1-Blue
    Lamp1 (561,492 48x43), variable: PLC_PRG.pos4, style: Lamp-Lamp1-Blue
    Lamp1 (508,492 48x43), variable: PLC_PRG.pos5, style: Lamp-Lamp1-Blue
    Lamp1 (456,492 48x43), variable: PLC_PRG.pos6, style: Lamp-Lamp1-Blue
    Lamp1 (403,492 48x43), variable: PLC_PRG.pos7, style: Lamp-Lamp1-Blue
    Lamp1 (720,492 48x43), variable: PLC_PRG.pos1, style: Lamp-Lamp1-Blue
    Lamp1 (351,492 48x43), variable: PLC_PRG.pos8, style: Lamp-Lamp1-Blue
    Lamp1 (298,492 48x43), variable: PLC_PRG.pos9, style: Lamp-Lamp1-Blue
    Label (438,144 175x42), "OCUPACION"
    Label (766,493 20x42), "1"
    Label (765,376 20x42), "19"
    Label (766,263 20x42), "37"
    Label (270,437 20x42), "18"
    Label (269,322 20x42), "36"
    Label (270,209 20x42), "54"
    Textfield (431,627 150x30), "%i", text variable: PLC_PRG.CNT_TOTAL.CV
    Label (431,606 150x30), "TOTAL MOVIMIENTOS"
    Lamp1 (157,538 50x41), variable: PLC_PRG.deteccion_pieza_robot_cart, style: Lamp-Lamp1-Yellow
    Label (106,509 150x30), "PIEZA EN CARTESIANO"
    Rectangle (103,430 156x73)
    Lamp1 (157,455 50x41), variable: PLC_PRG.SENSOR_piezas_cinta, style: Lamp-Lamp1-Yellow
    Label (105,136 150x30), "SISTEMA ON"
    Textfield (432,716 150x30), "%i", text variable: GVL.POSICION
    Label (432,695 150x30), "SIGUIENTE UBICACION"
    Table (822,164 278x403), data array: PLC_PRG.REGISTRO
        p1128707560: PLC_PRG.POS
        p3854506369: PLC_PRG.REGISTRO[INDEX]
        p1014161805: 55 - 1 + 1
    Rectangle (105,602 156x73)
    Lamp1 (159,627 50x41), variable: NOT PLC_PRG.At_load, style: Lamp-Lamp1-Yellow
    Label (108,598 150x30), "PIEZA EN TRASLO"
    Label (106,425 150x30), "PIEZA EN ROBOT"
    Label (857,133 199x30), "ENTRADAS/POSICION"
    Label (270,265 20x42), "45"
    Label (270,377 20x42), "27"
    Label (271,491 20x42), "9"
    Label (766,439 20x42), "10"
    Label (766,323 20x42), "28"
    Label (766,208 20x42), "46"
    Lamp1 (497,65 50x41), variable: PLC_PRG.ALARMA_ACTIVA, style: Lamp-Lamp1-Red
    Label (445,35 150x30), "ALARMA"
END_VISUALIZATION
